// Mitsubishi GX Works2 project: theori2   PLC: FX3G

// global labels: Global1
VAR_GLOBAL CONSTANT
  workTime : INT := 50;
END_VAR
VAR_GLOBAL
  endWorkTimer AT TC1 : BOOL;
  under950KG AT X001 : BOOL;
  endWorkTimer1 AT TS1 : BOOL;
  startButton AT X007 : BOOL;
  buttonPresed AT M1 : BOOL;
  OnProgress AT Y007 : BOOL;
  resetTimer AT X010 : BOOL;
  fictiveLamp1 AT Y001 : BOOL;
  TimerHolder AT M3 : BOOL;
  reached950KG AT X001 : BOOL;
  finishCounting AT Y001 : BOOL;
  boatIsEmpty AT X005 : BOOL;
  someoneIsNear AT X006 : BOOL;
  ExitGate AT Y000 : BOOL;
END_VAR

// task Task_01 (event TRUE, interval 0, priority 31): POU_01

PROGRAM POU_01
(* structured ladder/FBD written out as ST: instructions are called as NAME(EN, inputs, outputs); _pN, _eN, _tN stand for wires *)
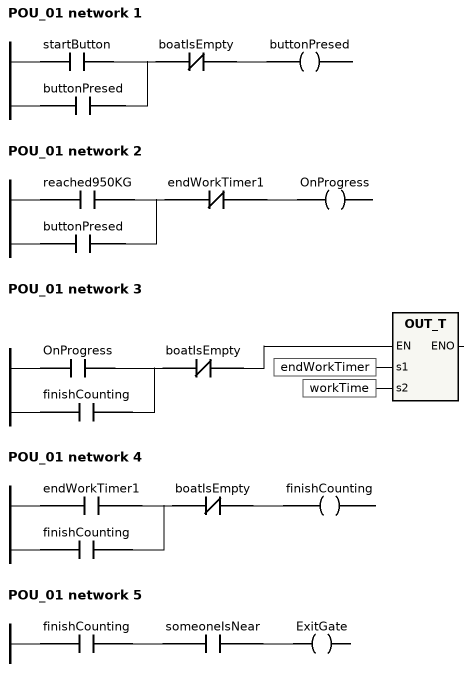
(* network 1 *)
buttonPresed := (startButton OR buttonPresed) AND NOT boatIsEmpty;
(* network 2 *)
OnProgress := (reached950KG OR buttonPresed) AND NOT endWorkTimer1;
(* network 3 *)
OUT_T((OnProgress OR finishCounting) AND NOT boatIsEmpty, endWorkTimer, workTime);
(* network 4 *)
finishCounting := (endWorkTimer1 OR finishCounting) AND NOT boatIsEmpty;
(* network 5 *)
ExitGate := finishCounting AND someoneIsNear;
END_PROGRAM
